{attribute 'reflection'}
FUNCTION_BLOCK FB_ReadTc3Events2 EXTENDS FB_ReadTc3Events
VAR_INPUT
	bClearLoggedTable : BOOL;
END_VAR

VAR_OUTPUT
	LoggedEvents : ARRAY[1..80] OF ST_ReadEventW;
END_VAR

VAR
	{attribute 'instance-path'}
	{attribute 'noinit'}
	sPath			   : T_MAXSTRING;
	CallReadTc3Events2 : NT_StartProcess;
	DeviceInfo		   : FB_GetDeviceIdentificationEx;
	Init			   : BOOL := TRUE;
	fbArgsFormat	   : FB_FormatString2;
	ReadTc3Events2Args : T_MAXSTRING;
	
	
	//Win32Events		   : FB_TcMessage;
END_VAR

VAR CONSTANT
	ArgsFormat : T_MAXSTRING := 'ReadTc3Events2.dll --symbolpath %s --languageid %d --datetimeformat %d ';
END_VAR

SUPER^();
IF bClearLoggedTable THEN
	MEMSET(ADR(LoggedEvents), 0, SIZEOF(LoggedEvents));
END_IF

IF Init THEN
	DeviceInfo(bExecute := TRUE, sNetId := '');
	IF NOT DeviceInfo.bBusy THEN
		DeviceInfo(bExecute := FALSE);

		//Set paths based on target system OS
		IF DeviceInfo.stDevIdent.strImageOsName = 'TwinCAT/BSD' THEN
			CallReadTc3Events2.PATHSTR := '/usr/local/bin/dotnet'; //doas pkg install dotnet
			CallReadTc3Events2.DIRNAME := '/usr/local/etc/TwinCAT/3.1/Components/Plc/ReadTc3Events2';
		END_IF

		Init := FALSE;
	END_IF
END_IF

CallReadTc3Events2(NETID := '', COMNDLINE := ReadTc3Events2Args);

//FB_Init is always available implicitly and it is used primarily for initialization.

//The return value is not evaluated. For a specific influence, you can also declare the

//methods explicitly and provide additional code there with the standard initialization

//code. You can evaluate the return value.
METHOD FB_Init : BOOL
VAR_INPUT
	bInitRetains : BOOL; // TRUE: the retain variables are initialized (reset warm / reset cold)
	bInCopyCode	 : BOOL; // TRUE: the instance will be copied to the copy code afterward (online change)   
END_VAR

VAR
	sDot		  : STRING(2) := '.';
	sEmpty		  : STRING(1) := ''; // replacement = empty
	sTmpOut		  : STRING(255);	 // <-- set >= max length of sPath
	nFirstPos	  : UDINT;
	nSecondPosRel : UDINT;
	nSecondPosAbs : UDINT;
	nRemoveLen	  : UDINT;
	bOk			  : BOOL;
END_VAR
//Win32Events.CreateEx(TC_EVENTS.Win32EventClass.ERROR_SUCCESS,0); /

//Use the Win32EventClass - so event logger knows about Win32EventClass GUID. Used by the dotnet application
TC_EVENTS.Win32EventClass;


//Trim the project name, and PLC name from the function block instance path
// Find first dot
nFirstPos := FIND2(ADR(sPath), ADR(sDot));

IF nFirstPos > 0 THEN
    // Find second dot by searching from just after the first one
    nSecondPosRel := FIND2(ADR(sPath) + nFirstPos, ADR(sDot));

    IF nSecondPosRel > 0 THEN
        // Convert relative position to absolute (1-based indexing)
        nSecondPosAbs := nFirstPos + nSecondPosRel;

        // Remove everything from start through the second dot
        nRemoveLen := nSecondPosAbs;

        bOk := REPLACE2(
            pSrcString    := ADR(sPath),
            pInsertString := ADR(sEmpty),
            pDstString    := ADR(sTmpOut),
            nDstSize      := SIZEOF(sTmpOut),
            nLen          := nRemoveLen,
            nPos          := 1
        );

        // Overwrite sPath with the result (even if truncated)
        sPath := CONCAT(sTmpOut,'.LoggedEvents');
    END_IF
END_IF
END_METHOD

//A rising edge on the input parameter bExec triggers the Read procedure. 

//The asynchronous process is terminated as soon as the reference bExec is set back to FALSE from the method. 

//When the process ends, the return value of the method indicates whether the call to ReadTc3Events2 was successful (TRUE) or failed (FALSE) for the duration of one call.
METHOD ReadLoggedEvents : BOOL;
VAR_INPUT
	bExec : REFERENCE TO BOOL;
END_VAR

VAR_OUTPUT
	hrErrorCode : HRESULT;
END_VAR

VAR_INST
	Step : UDINT;
END_VAR
CASE Step OF
	0:
		fbArgsFormat(pFormatString := ADR(ArgsFormat),
					 arg1		   := F_STRING(sPath),
					 arg2		   := F_DINT(THIS^.nLanguageID),
					 arg3		   := F_INT(THIS^.eDateAndTimeFormat),
					 pDstString	   := ADR(ReadTc3Events2Args),
					 nDstSize	   := SIZEOF(ReadTc3Events2Args));

		IF fbArgsFormat.bError THEN
			bExec			 := FALSE;
			ReadLoggedEvents := FALSE;
			hrErrorCode		 := fbArgsFormat.nErrId;
			RETURN;
		END_IF

		CallReadTc3Events2.START := TRUE;
		Step					 := 10;

	10:
		IF NOT CallReadTc3Events2.BUSY THEN
			IF NOT CallReadTc3Events2.ERR THEN
				hrErrorCode		 := 0;
				ReadLoggedEvents := TRUE;
			ELSE
				hrErrorCode		 := CallReadTc3Events2.ERRID;
				ReadLoggedEvents := FALSE;
			END_IF

			bExec					 := FALSE;
			Step					 := 0;
			CallReadTc3Events2.START := FALSE;
		END_IF
END_CASE
END_METHOD

END_FUNCTION_BLOCK

(* stored: Version 1.1.0.1
   POU FB_ReadTc3Events2: Id {5a6edfd8-5abe-4422-80aa-514948601d1b}, SpecialFunc None
   Method FB_Init: Id {518a7732-9a1b-4fc5-8f94-24f44370f21e}
   Method ReadLoggedEvents: Id {936688d8-92ba-4ae8-8c66-ec3f8ec0b489} *)
